# EPICS substitutions: MOXA12XX/MOXA12XX-IOC-01App/Db/moxa_e1262_PVs.substitutions
file "IBEX_PVs_channels.template" {

pattern {NAME, P, ASYNPORT, OLDFNCTN, CHAN, NEWFNCTN}

# Scaled values
{"\$(NAME)", "\$(P)", "\$(ASYNPORT)", "AI", "0", "TEMP:RBV"}
{"\$(NAME)", "\$(P)", "\$(ASYNPORT)", "AI", "1", "TEMP:RBV"}
{"\$(NAME)", "\$(P)", "\$(ASYNPORT)", "AI", "2", "TEMP:RBV"}
{"\$(NAME)", "\$(P)", "\$(ASYNPORT)", "AI", "3", "TEMP:RBV"}
{"\$(NAME)", "\$(P)", "\$(ASYNPORT)", "AI", "4", "TEMP:RBV"}
{"\$(NAME)", "\$(P)", "\$(ASYNPORT)", "AI", "5", "TEMP:RBV"}
{"\$(NAME)", "\$(P)", "\$(ASYNPORT)", "AI", "6", "TEMP:RBV"}
{"\$(NAME)", "\$(P)", "\$(ASYNPORT)", "AI", "7", "TEMP:RBV"}
